Fanuc KAREL source: ko00068.KL

-- PROVISIONAL review KL for V1013-1; original PC SHA256 77a37354c85a3ebab0bcd83fe9832e664929548576a49c73cf72eafd2562e491
-- Incomplete behavior may be omitted. Consult companion uncertainty JSON. Do not deploy.
PROGRAM KO00068
%NOLOCKGROUP
BEGIN
  -- UNRESOLVED_PC offsets 5-12; opcodes 9D,23
  -- UNRESOLVED_PC offsets 17-63; opcodes 27,22,1C,22,1C,22,31,7E,4A
  -- UNRESOLVED_PC offsets 68-72; opcodes 7F
END KO00068
